FUNCTION_BLOCK EL4122
VAR
	_io : EL4xx2_Data;
	{attribute addProperty Name "WcState"}
	_wcState : WcStateBase;
	{attribute addProperty Name "Info data"}
	_infoData : InfoDataAds;
END_VAR

PROPERTY IO : REFERENCE TO EL4xx2_Data
GET
IO REF= _io;
END_GET
END_PROPERTY

PROPERTY WcState : REFERENCE TO WcStateBase
GET
WcState REF= _wcState;
END_GET
END_PROPERTY

END_FUNCTION_BLOCK

(* stored: Version 1.1.0.1, ProductVersion 3.1.4024.9
   POU EL4122: Id {a8cd7283-933b-0b15-147d-b41ebfb31b53}, SpecialFunc None
   Property IO: Id {1aeec262-7215-09d0-3150-523aef6893f6}
   Get Get: Id {723bc55c-b0b6-0d9b-3929-40d410b88bb1}
   Property WcState: Id {8a82f277-5d7c-05e5-3f6d-b89ec74567e0}
   Get Get: Id {1c9209b4-2bbe-0ee4-0e31-0ed22ab31e24} *)
